// TwinCAT 3 PLC project tins
// ProgramVersion: 3.1.4023.0
// libraries:
//   ESO LDC Lamp Library, * (ESO)
//   ESO LDC Motor Library, * (ESO)
//   ESO LDC Piezo Library, * (ESO)
//   ESO LDC Shutter Library, * (ESO)
//   ESO LDC Timer Library, * (ESO)
//   Tc2_Standard, * (Beckhoff Automation GmbH)
//   Tc2_System, * (Beckhoff Automation GmbH)
//   Tc3_Module, * (Beckhoff Automation GmbH)
//   VisuDialogs, * (System)
//   VisuSymbols,3.5.10.0,System
// project tree:
//   / GlobalTextList.TcGTLO, PlcTask.TcTTO, Visualization Manager.TcVMO (not stored)
//   POUs/ MAIN.TcPOU
//   VISUs/ adc1.TcVIS, drot1.TcVIS, lamp1.TcVIS, shutter1.TcVIS
// real-time tasks:
//   TASK PlcTask: cycle T#10ms, priority 20, ADS port 350
// motion (NC):
//   TASK NC-Task 1 SAF: cycle T#2ms, priority 4, ADS port 501
//   TASK NC-Task 1 SVB: cycle T#10ms, priority 8, ADS port 511
//   AXIS Motor1 (id 1)
//     OtherSettings: AllowMotionCmdToSlave=true
//     encoder EncType=1
//     drive DrvType=5
//       Analog: TorqueSetpointScale=10, ScaleFactorActTorque=0.1
//       TimeComp: TaskDelayCycles=1
//     controller CtrType=1
//       CtrPara: PriorControlFactor=1
//         Observer: BandWidth=20
//   AXIS Motor2 (id 2)
//     OtherSettings: AllowMotionCmdToSlave=true
//     encoder EncType=1
//     drive DrvType=5
//       Analog: TorqueSetpointScale=10, ScaleFactorActTorque=0.1
//       TimeComp: TaskDelayCycles=1
//     controller CtrType=1
//       CtrPara: PriorControlFactor=1
//         Observer: BandWidth=20
//   AXIS AdcMotor1 (id 3)
//     OtherSettings: AllowMotionCmdToSlave=true
//     encoder EncType=1
//     drive DrvType=5
//       Analog: TorqueSetpointScale=10, ScaleFactorActTorque=0.1
//       TimeComp: TaskDelayCycles=1
//     controller CtrType=1
//       CtrPara: PriorControlFactor=1
//         Observer: BandWidth=20
//   AXIS AdcMotor2 (id 4)
//     OtherSettings: AllowMotionCmdToSlave=true
//     encoder EncType=1
//     drive DrvType=5
//       Analog: TorqueSetpointScale=10, ScaleFactorActTorque=0.1
//       TimeComp: TaskDelayCycles=1
//     controller CtrType=1
//       CtrPara: PriorControlFactor=1
//         Observer: BandWidth=20
//   AXIS DrotMotor (id 5)
//     OtherSettings: AllowMotionCmdToSlave=true
//     encoder EncType=1
//     drive DrvType=5
//       Analog: TorqueSetpointScale=10, ScaleFactorActTorque=0.1
//       TimeComp: TaskDelayCycles=1
//     controller CtrType=1
//       CtrPara: PriorControlFactor=1
//         Observer: BandWidth=20
// variable links:
//   tins/tins Instance <-> NC-Task 1 SAF/Axes/AdcMotor1
//     PlcTask Inputs/MAIN.adc1.motor1.Axis.NcToPlc <-> Outputs/ToPlc
//     PlcTask Outputs/MAIN.adc1.motor1.Axis.PlcToNc <-> Inputs/FromPlc
//   tins/tins Instance <-> NC-Task 1 SAF/Axes/AdcMotor2
//     PlcTask Inputs/MAIN.adc1.motor2.Axis.NcToPlc <-> Outputs/ToPlc
//     PlcTask Outputs/MAIN.adc1.motor2.Axis.PlcToNc <-> Inputs/FromPlc
//   tins/tins Instance <-> NC-Task 1 SAF/Axes/DrotMotor
//     PlcTask Inputs/MAIN.drot1.motor.Axis.NcToPlc <-> Outputs/ToPlc
//     PlcTask Outputs/MAIN.drot1.motor.Axis.PlcToNc <-> Inputs/FromPlc
//   tins/tins Instance <-> NC-Task 1 SAF/Axes/Motor1
//     PlcTask Inputs/MAIN.Motor1.Axis.NcToPlc <-> Outputs/ToPlc
//     PlcTask Outputs/MAIN.Motor1.Axis.PlcToNc <-> Inputs/FromPlc
//   tins/tins Instance <-> NC-Task 1 SAF/Axes/Motor2
//     PlcTask Inputs/MAIN.Motor2.Axis.NcToPlc <-> Outputs/ToPlc
//     PlcTask Outputs/MAIN.Motor2.Axis.PlcToNc <-> Inputs/FromPlc
//   tins/tins Instance <-> tins/tins Instance
//     PlcTask Inputs/MAIN.Lamp1.i_bFault <-> PlcTask Outputs/MAIN.SIM_Lamp1.q_bFault
//     PlcTask Inputs/MAIN.Lamp1.i_bOn <-> PlcTask Outputs/MAIN.SIM_Lamp1.q_bOn
//     PlcTask Inputs/MAIN.Motor1.i_nCouplerState <-> PlcTask Outputs/MAIN.SIM_Motor1.q_nCouplerState
//     PlcTask Inputs/MAIN.Motor1.switches <-> PlcTask Outputs/MAIN.SIM_Motor1.switches
//     PlcTask Inputs/MAIN.Motor2.switches <-> PlcTask Outputs/MAIN.SIM_Motor2.switches
//     PlcTask Inputs/MAIN.Motor2.i_bBrake_Stat <-> PlcTask Outputs/MAIN.SIM_Motor2.q_bBrake_Stat
//     PlcTask Inputs/MAIN.Piezo1.i_nCouplerState <-> PlcTask Outputs/MAIN.SIM_Piezo1.q_nCouplerState
//     PlcTask Inputs/MAIN.SIM_Motor2.i_bBrake_Ctrl <-> PlcTask Outputs/MAIN.Motor2.q_bBrake_Ctrl
//     PlcTask Inputs/MAIN.SIM_Piezo1.i_nSignal <-> PlcTask Outputs/MAIN.Piezo1.q_nCtrl
//     PlcTask Inputs/MAIN.Shutter1.i_bFault <-> PlcTask Outputs/MAIN.SIM_Shutter1.q_bFault
//     PlcTask Inputs/MAIN.Shutter1.i_bOpen <-> PlcTask Outputs/MAIN.SIM_Shutter1.q_bOpen
//     PlcTask Inputs/MAIN.adc1.i_ccs_data <-> PlcTask Outputs/MAIN.ccs_sim.q_ccs_data
//     PlcTask Inputs/MAIN.adc1.motor1.i_bBrake_Stat <-> PlcTask Outputs/MAIN.SIM_adc_motor1.q_bBrake_Stat
//     PlcTask Inputs/MAIN.adc1.motor1.switches <-> PlcTask Outputs/MAIN.SIM_adc_motor1.switches
//     PlcTask Inputs/MAIN.drot1.motor.i_nCouplerState <-> PlcTask Outputs/MAIN.SIM_drot_motor.q_nCouplerState
//     PlcTask Outputs/MAIN.Lamp1.q_bSwitch <-> PlcTask Inputs/MAIN.SIM_Lamp1.i_bSwitch
//     PlcTask Outputs/MAIN.Lamp1.q_nIntensity <-> PlcTask Inputs/MAIN.Lamp1.i_nOn
//     PlcTask Outputs/MAIN.Motor1.q_bBrake_Ctrl <-> PlcTask Inputs/MAIN.SIM_Motor1.i_bBrake_Ctrl
//     PlcTask Outputs/MAIN.SIM_Lamp1.q_nCouplerState <-> PlcTask Inputs/MAIN.Lamp1.i_nCouplerState
//     PlcTask Outputs/MAIN.SIM_Motor1.q_bBrake_Stat <-> PlcTask Inputs/MAIN.Motor1.i_bBrake_Stat
//     PlcTask Outputs/MAIN.SIM_Motor2.q_nCouplerState <-> PlcTask Inputs/MAIN.Motor2.i_nCouplerState
//     PlcTask Outputs/MAIN.SIM_Piezo1.q_nSignal <-> PlcTask Inputs/MAIN.Piezo1.i_nActVal_Int16
//     PlcTask Outputs/MAIN.SIM_Shutter1.q_bClosed <-> PlcTask Inputs/MAIN.Shutter1.i_bClosed
//     PlcTask Outputs/MAIN.SIM_Shutter1.q_nCouplerState <-> PlcTask Inputs/MAIN.Shutter1.i_nCouplerState
//     PlcTask Outputs/MAIN.SIM_adc_motor1.q_nCouplerState <-> PlcTask Inputs/MAIN.adc1.motor1.i_nCouplerState
//     PlcTask Outputs/MAIN.SIM_adc_motor2.q_nCouplerState <-> PlcTask Inputs/MAIN.adc1.motor2.i_nCouplerState
//     PlcTask Outputs/MAIN.SIM_adc_motor2.q_bBrake_Stat <-> PlcTask Inputs/MAIN.adc1.motor2.i_bBrake_Stat
//     PlcTask Outputs/MAIN.SIM_adc_motor2.switches <-> PlcTask Inputs/MAIN.adc1.motor2.switches
//     PlcTask Outputs/MAIN.SIM_drot_motor.q_bBrake_Stat <-> PlcTask Inputs/MAIN.drot1.motor.i_bBrake_Stat
//     PlcTask Outputs/MAIN.SIM_drot_motor.switches <-> PlcTask Inputs/MAIN.drot1.motor.switches
//     PlcTask Outputs/MAIN.Shutter1.q_bSwitch <-> PlcTask Inputs/MAIN.SIM_Shutter1.i_bSwitch
//   tins/tins Instance <-> TcCOM Objects/Object1 (trkModule)
//     PlcTask Inputs/MAIN.adc1.i_trk_data <-> Outputs/TrackingData
//     PlcTask Inputs/MAIN.ccs_sim.i_trk_data <-> Outputs/TrackingData
//     PlcTask Inputs/MAIN.drot1.i_ccs_data <-> Outputs/TrackingData/computation
//     PlcTask Inputs/MAIN.drot1.i_trk_data <-> Outputs/TrackingData
//     PlcTask Outputs/MAIN.timer.q_timeInfo <-> Inputs/TimeInfo
//   tins/tins Instance <-> TcCOM Objects/Object2 (trkParams)
//     PlcTask Outputs/MAIN.ccs_sim.q_ccs_data <-> Inputs/CcsData
//     PlcTask Outputs/MAIN.timer.q_timeInfo <-> Inputs/TimeInfo
//   TcCOM Objects/Object1 (trkModule) <-> TcCOM Objects/Object2 (trkParams)
//     Inputs/SlaParams <-> Outputs/SlaParams

CONFIGURATION tins
    RESOURCE PLC ON TwinCAT3
        TASK PlcTask(INTERVAL := T#10ms, PRIORITY := 20);
        PROGRAM MAIN WITH PlcTask : MAIN;
    END_RESOURCE
END_CONFIGURATION

// ---- POUs/MAIN.TcPOU
PROGRAM MAIN
VAR
	{attribute 'OPC.UA.DA':='1'}
	Shutter1:		FB_SHUTTER;
	{attribute 'OPC.UA.DA':='1'}
	Lamp1:		FB_LAMP;
	{attribute 'OPC.UA.DA':='1'}
	Piezo1:		FB_PIEZO_EXAMPLE;	// Piezo #1
	
	{attribute 'OPC.UA.DA':='1'}
	Motor1:		FB_MOTOR;		
	{attribute 'OPC.UA.DA':='1'}
	Motor2:		FB_MOTOR;		
	{attribute 'OPC.UA.DA':='1'}
	adc1:		FB_MA_ADC;
	
    {attribute 'OPC.UA.DA':='1'}
	drot1:       FB_MA_DROT;
	
	ccs_sim:	FB_CCS_SIM;
	timer: FB_TIME;
	{attribute 'OPC.UA.DA':='1'}
	SIM_Shutter1:	FB_SIM_SHUTTER;
	{attribute 'OPC.UA.DA':='1'}
	SIM_Lamp1:	FB_SIM_LAMP;
	{attribute 'OPC.UA.DA':='1'}
	SIM_Piezo1:	FB_SIM_PIEZO;		// Simulator for Piezo #1 (if simulated)
	
	{attribute 'OPC.UA.DA':='1'}
	SIM_Motor1:	FB_SIM_MOTOR;
	{attribute 'OPC.UA.DA':='1'}
	SIM_Motor2:	FB_SIM_MOTOR;
	{attribute 'OPC.UA.DA':='1'}
	SIM_adc_motor1:	FB_SIM_MOTOR;
	{attribute 'OPC.UA.DA':='1'}
	SIM_adc_motor2:	FB_SIM_MOTOR;
	{attribute 'OPC.UA.DA':='1'}
	SIM_drot_motor:	FB_SIM_MOTOR;
END_VAR

Shutter1(in_sName:='Shutter001');
Lamp1(in_sName:='Lamp001', in_nTimeout:=5000);

Piezo1(in_sName:='Piezo001', in_nNumAxes:=3);

Motor1(sName:='Motor1',nNOVRAM_DevId:=0);
Motor2(sName:='Motor2',nNOVRAM_DevId:=0);

// ADC
adc1(sName:='ADC', sMotorAdc1:= 'ADC1', sMotorAdc2:= 'ADC2');
SIM_adc_motor1(ptrCfg:=ADR(adc1.motor1.cfg), 	ptrStat:=ADR(adc1.motor1.stat));
SIM_adc_motor2(ptrCfg:=ADR(adc1.motor2.cfg), 	ptrStat:=ADR(adc1.motor2.stat));

// DROT
//
drot1(sName:='DROT', sMotorName:= 'DrotMotor', nNOVRAM_DevId:=0);
SIM_drot_motor(ptrCfg:=ADR(drot1.motor.cfg), ptrStat:=ADR(drot1.motor.stat));

ccs_sim();

timer();

// Simulators
SIM_Shutter1(ptrDev := ADR(Shutter1));
SIM_Lamp1(ptrDev:=ADR(Lamp1));
SIM_Piezo1();

SIM_Motor1(ptrCfg:=ADR(Motor1.cfg), 	ptrStat:=ADR(Motor1.stat));
SIM_Motor2(ptrCfg:=ADR(Motor2.cfg), 	ptrStat:=ADR(Motor2.stat));

END_PROGRAM

// ---- VISUs/adc1.TcVIS
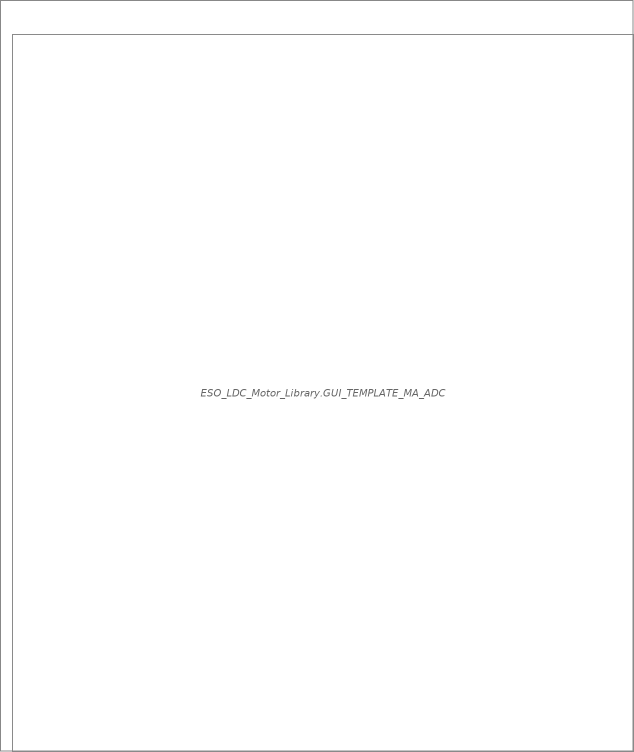
VISUALIZATION adc1  // 634x752
    Frame (12,34 622x718)
        shows ESO_LDC_Motor_Library.GUI_TEMPLATE_MA_ADC(m_DeviceName := 'ADC1', m_Instance := MAIN.adc1)
END_VISUALIZATION

// ---- VISUs/drot1.TcVIS
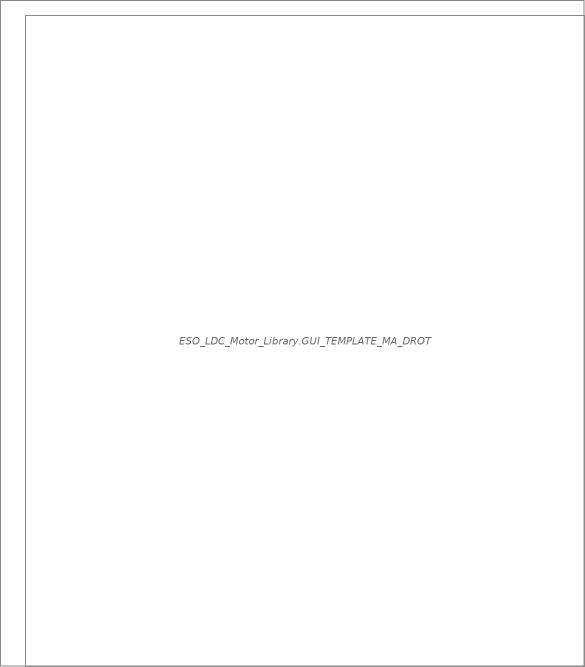
VISUALIZATION drot1  // 585x667
    Frame (25,15 560x652)
        shows ESO_LDC_Motor_Library.GUI_TEMPLATE_MA_DROT(m_DeviceName := 'drot1', m_Instance := MAIN.drot1)
END_VISUALIZATION

// ---- VISUs/lamp1.TcVIS
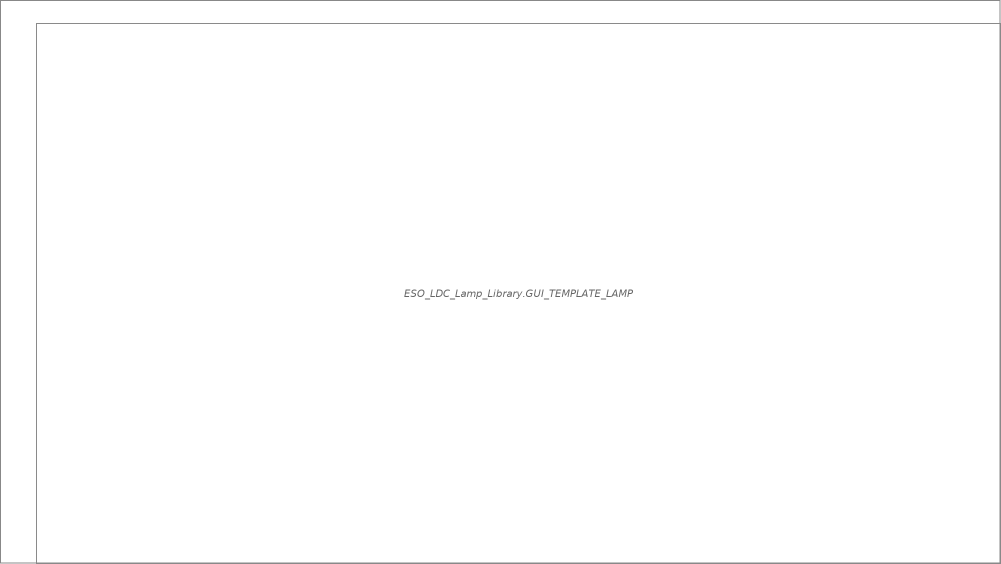
VISUALIZATION lamp1  // 1001x564
    Frame (36,23 965x541)
        shows ESO_LDC_Lamp_Library.GUI_TEMPLATE_LAMP(m_Instance := MAIN.Lamp1)
END_VISUALIZATION

// ---- VISUs/shutter1.TcVIS
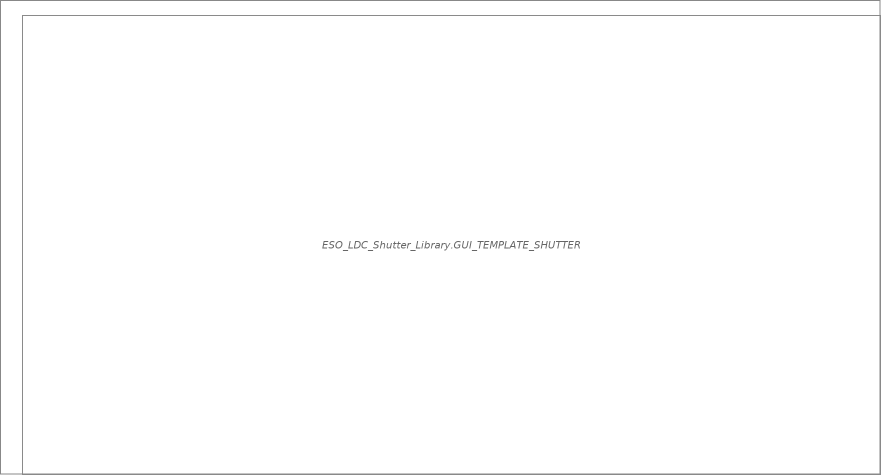
VISUALIZATION shutter1  // 881x475
    Frame (22,15 859x460)
        shows ESO_LDC_Shutter_Library.GUI_TEMPLATE_SHUTTER(m_Instance := MAIN.Shutter1)
END_VISUALIZATION
